// TwinCAT 3 PLC project LAB7_PLC
// ProgramVersion: 3.1.4023.0
// libraries:
//   Tc2_Standard, * (Beckhoff Automation GmbH)
//   Tc2_System, * (Beckhoff Automation GmbH)
//   Tc3_Module, * (Beckhoff Automation GmbH)
// project tree:
//   DUTs/ E_Crane_Status.TcDUT, E_Mode.TcDUT, ST_pPistonStroke.TcDUT
//   / GlobalTextList.TcGTLO, PlcTask.TcTTO, Visualization Manager.TcVMO (not stored)
//   GVLs/ HMI.TcGVL, input.TcGVL, output.TcGVL, parameter.TcGVL
//   POUs/ MAIN.TcPOU, Set_New_Max_Stroke.TcPOU
//   VISUs/ CraneHMI.TcVIS
// real-time tasks:
//   TASK PlcTask: cycle T#10ms, priority 20, ADS port 350

CONFIGURATION LAB7_PLC
    RESOURCE PLC ON TwinCAT3
        TASK PlcTask(INTERVAL := T#10ms, PRIORITY := 20);
        PROGRAM MAIN WITH PlcTask : MAIN;
    END_RESOURCE
END_CONFIGURATION

// ---- DUTs/E_Crane_Status.TcDUT
{attribute 'qualified_only'}
{attribute 'strict'}
TYPE E_Crane_Status :
(
	Running,
	Unnabled,
	Ready
);
END_TYPE

// ---- DUTs/E_Mode.TcDUT
{attribute 'qualified_only'}
{attribute 'strict'}
TYPE E_Mode :
(
	Auto,
	Manual 
);
END_TYPE

// ---- DUTs/ST_pPistonStroke.TcDUT
TYPE ST_pPistonStroke :
STRUCT
	rCylinderStrokeMax : REAL := 1.0;
	rCylinderStrokeMin : REAL := 0.0;
END_STRUCT
END_TYPE

// ---- GVLs/HMI.TcGVL
{attribute 'qualified_only'}
VAR_GLOBAL
	sPistonEndStopMessage : STRING;
END_VAR

// ---- GVLs/input.TcGVL
{attribute 'qualified_only'}
VAR_GLOBAL
	bEnableSwitch : BOOL;
	bModeSwitch : BOOL;
	bStartSwitch : BOOL;	
	bSetNewMaxStrokeSwitch: BOOL;
	rSetInputMaxStroke : REAL;










END_VAR

// ---- GVLs/output.TcGVL
{attribute 'qualified_only'}
VAR_GLOBAL
	
	bRunningLight : BOOL;
	rCylinderVel : REAL;
	rCylinderPos : REAL;
	


	
END_VAR

// ---- GVLs/parameter.TcGVL
{attribute 'qualified_only'}
VAR_GLOBAL
	
	rRefCylinderVel : REAL;
	rRefCylinderPos : REAL;
	rAutoTime : REAL;
	rCycleTime : REAL := 0.01;
	stStrokeRange : ST_pPistonStroke;
	rRunTime : REAL;
	rInitialStrokePosition : REAL;
END_VAR

// ---- POUs/MAIN.TcPOU
PROGRAM MAIN
VAR
	eStatus : E_CRANE_STATUS;
	eMode : E_Mode;
	aEndStopMessages : ARRAY[0..2] OF STRING := ['END STOP NOT ACTIVE' , 'PISTON HAS REACHED UPPER END STOP', 'PISTON HAS REACHED LOWER END STOP'];
	sEndStopMessage : STRING;
END_VAR


IF input.bEnableSwitch = FALSE THEN
output.bRunningLight := FALSE;
input.bStartSwitch := FALSE;
output.rCylinderVel := 0;
eStatus := E_Crane_Status.Unnabled;
END_IF



// Status message on HMI
IF input.bEnableSwitch = TRUE AND input.bStartSwitch = FALSE THEN
	eStatus := E_Crane_Status.Ready;
END_IF





IF input.bStartSwitch = FALSE THEN
	output.bRunningLight := FALSE;
	parameter.rRunTime := 0;
ELSIF input.bStartSwitch = TRUE THEN
	output.bRunningLight := TRUE;
	parameter.rRunTime := parameter.rRunTime + parameter.rCycleTime;
	eStatus := E_Crane_Status.Running;
END_IF





// Mode display on HMI
IF input.bModeSwitch = TRUE THEN
	eMode := E_mode.Auto;
ELSE
	eMode := E_Mode.Manual;
END_IF


// Set new max stroke
IF input.bSetNewMaxStrokeSwitch = TRUE THEN
	parameter.stStrokeRange.rCylinderStrokeMax :=Set_New_Max_Stroke(rNewMaxStroke := input.rSetInputMaxStroke);
	

input.bSetNewMaxStrokeSwitch := FALSE;
END_IF




// ENDSTOP MESSAGE
IF output.rCylinderPos >= parameter.stStrokeRange.rCylinderStrokeMax THEN
	sEndStopMessage := aEndStopMessages[1];
ELSIF output.rCylinderPos <= parameter.stStrokeRange.rCylinderStrokeMin THEN
	sEndstopMessage := aEndStopMessages[2];
ELSE
		sEndStopMessage := aEndStopMessages[0];
END_IF




// Manual Mode
IF input.bStartSwitch = TRUE AND input.bModeSwitch = FALSE THEN
	parameter.rAutoTime := 0;
	output.rCylinderPos := parameter.rRefCylinderPos;
END_IF




// AUTOMODE
IF input.bStartSwitch = TRUE
AND input.bModeSwitch = TRUE
THEN

	parameter.rInitialStrokePosition := parameter.rRefCylinderPos;
	
	// If stroke is maxed out:
	IF output.rCylinderPos >= parameter.stStrokeRange.rCylinderStrokeMax AND parameter.rRefCylinderVel > 0 THEN
		parameter.rAutoTime := 0;
		output.rCylinderVel := 0;
		
	
	// If piston is at bottom position:
	ELSIF output.rCylinderPos <= parameter.stStrokeRange.rCylinderStrokeMin AND parameter.rRefCylinderVel < 0 THEN
		parameter.rAutoTime := 0;
		output.rCylinderVel := 0;
		
	
	// When piston is between max and min:
	ELSE
		parameter.rAutoTime := parameter.rAutoTime + parameter.rCycleTime;
		output.rCylinderVel := parameter.rRefCylinderVel;
	
	END_IF
	
	output.rCylinderPos := parameter.rInitialStrokePosition + output.rCylinderVel * parameter.rAutoTime;
	parameter.rRefCylinderPos := output.rCylinderPos;
END_IF

END_PROGRAM

// ---- POUs/Set_New_Max_Stroke.TcPOU
FUNCTION Set_New_Max_Stroke : REAL
VAR_INPUT
	rNewMaxStroke : REAL;
END_VAR
VAR
END_VAR

IF rNewMaxStroke < -0.005 OR rNewMaxStroke > 0.005 THEN
	Set_New_Max_Stroke := 0;
ELSE
	Set_New_Max_Stroke := rNewMaxStroke;
END_IF

END_FUNCTION

// ---- GlobalTextList.TcGTLO
TEXTLIST GlobalTextList
  394 = '%0.1f'
  201 = '%1.1f'
  7 = '%1.2f'
  46 = '%1.3f'
  138 = '%f'
  76 = '%I'
  439 = '%i'
  336 = '%s'
  767 = 'ATUO'
  85 = 'Crane'
  330 = 'CYLINDER STROKE'
  503 = 'CYLINDER VELOCITY'
  988 = 'ENABLE'
  211 = 'MANUAL'
  712 = 'RUNNING'
  212 = 'Set New Value'
  473 = 'START'
  523 = 'TIME RUNNING'
END_TEXTLIST

// ---- VISUs/CraneHMI.TcVIS
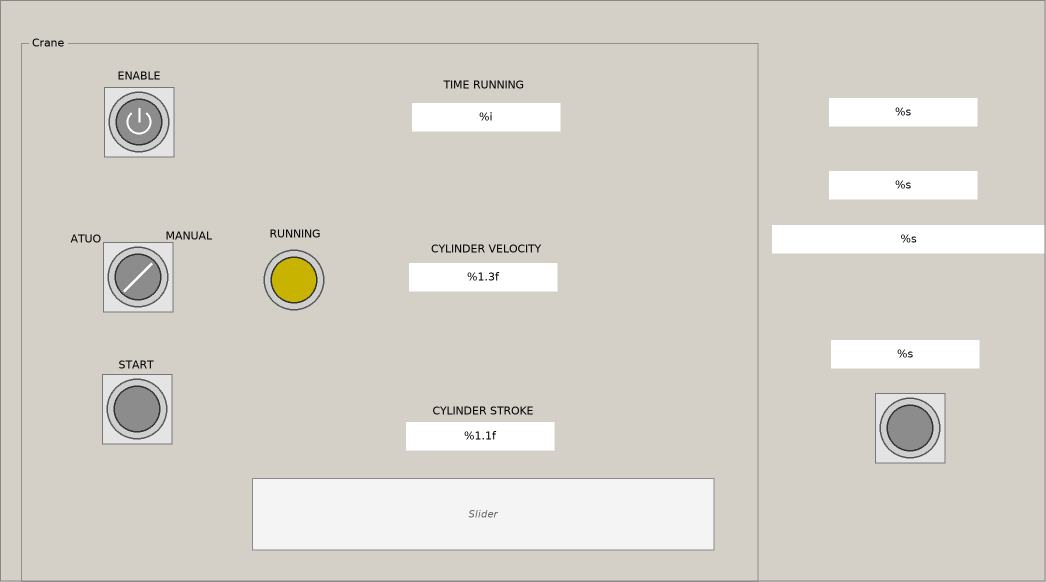
VISUALIZATION CraneHMI  // 1046x582
    Lamp1 (259,245 70x70), variable: output.bRunningLight, style: Lamp-Lamp1-Yellow
    PowerSwitch (104,87 70x70), variable: input.bEnableSwitch, behaviour: TOGGLE, style: Switch-PowerSwitch-Gray
    PushSwitch (102,374 70x70), variable: input.bStartSwitch, behaviour: TOGGLE, style: Switch-PushSwitch-Gray
    RotarySwitch (103,242 70x70), variable: input.bModeSwitch, behaviour: TOGGLE, style: Switch-RotarySwitch-Gray
    Label (114,221 150x30), "MANUAL"
    Label (220,219 150x30), "RUNNING"
    Label (61,350 150x30), "START"
    Label (11,224 150x30), "ATUO"
    Label (64,61 150x30), "ENABLE"
    Textfield (408,262 150x30), "%1.3f", text variable: output.rCylinderVel
    Textfield (405,421 150x30), "%1.1f", text variable: output.rCylinderPos
    Label (411,234 150x30), "CYLINDER VELOCITY"
    Label (408,396 150x30), "CYLINDER STROKE"
    Textfield (411,102 150x30), "%i", text variable: parameter.rRunTime
    Label (409,70 150x30), "TIME RUNNING"
    Slider (252,478 462x72), variable: parameter.rRefCylinderPos, scale 0..1
    GroupBox (21,35 737x547), "Crane"
    Textfield (828,97 150x30), "%s", text variable: MAIN.eStatus
    Textfield (828,170 150x30), "%s", text variable: MAIN.eMode
    Textfield (771,224 275x30), "%s", text variable: MAIN.sEndStopMessage
    Textfield (830,339 150x30), "%s", text variable: input.rSetInputMaxStroke
    PushSwitch (875,393 70x70), variable: input.bSetNewMaxStrokeSwitch, behaviour: TOGGLE, style: Switch-PushSwitch-Gray
END_VISUALIZATION
